// TIA Portal V20 export
DATA_BLOCK "instFB_MCDDataTransfer"   // DB5
// stored: InstanceOfName FB_MCDDataTransfer, InstanceOfType FB
"FB_MCDDataTransfer"
BEGIN
END_DATA_BLOCK
